{attribute 'GeneratedUsingTerminal: EL1259-0000-0016'}
{attribute addProperty BoxType "EL1259-0000-0016"}
{attribute addProperty Id "Output_event_state_1BOOL1Output_event_state_2BOOL1Output_event_state_3BOOL1Output_event_state_4BOOL1Output_event_state_5BOOL1Output_event_state_6BOOL1Output_event_state_7BOOL1Output_event_state_8BOOL1Output_event_state_9BOOL1Output_event_state_10BOOL1"}
{attribute addProperty CRC "2836416589"}
{attribute addProperty Size "10"}
TYPE Outputs_A910484D :
STRUCT
	{attribute addProperty Name "Output_event_state_1"}
	Output_event_state_1 : BOOL;
	{attribute addProperty Name "Output_event_state_2"}
	Output_event_state_2 : BOOL;
	{attribute addProperty Name "Output_event_state_3"}
	Output_event_state_3 : BOOL;
	{attribute addProperty Name "Output_event_state_4"}
	Output_event_state_4 : BOOL;
	{attribute addProperty Name "Output_event_state_5"}
	Output_event_state_5 : BOOL;
	{attribute addProperty Name "Output_event_state_6"}
	Output_event_state_6 : BOOL;
	{attribute addProperty Name "Output_event_state_7"}
	Output_event_state_7 : BOOL;
	{attribute addProperty Name "Output_event_state_8"}
	Output_event_state_8 : BOOL;
	{attribute addProperty Name "Output_event_state_9"}
	Output_event_state_9 : BOOL;
	{attribute addProperty Name "Output_event_state_10"}
	Output_event_state_10 : BOOL;
END_STRUCT
END_TYPE

(* stored: Version 1.2.0.0, ProductVersion 3.1.4024.9
   DUT Outputs_A910484D: Id {72ba418d-f582-48c6-9809-3b563912ceba} *)
